SYSTEM Test Reader
  (* Version 1.0, 2005-06-27, Goran Cengic, Chalmers *)
  DEVICE Test Device : DeviceType_not_used
    RESOURCE TestResource : ResourceType_not_used
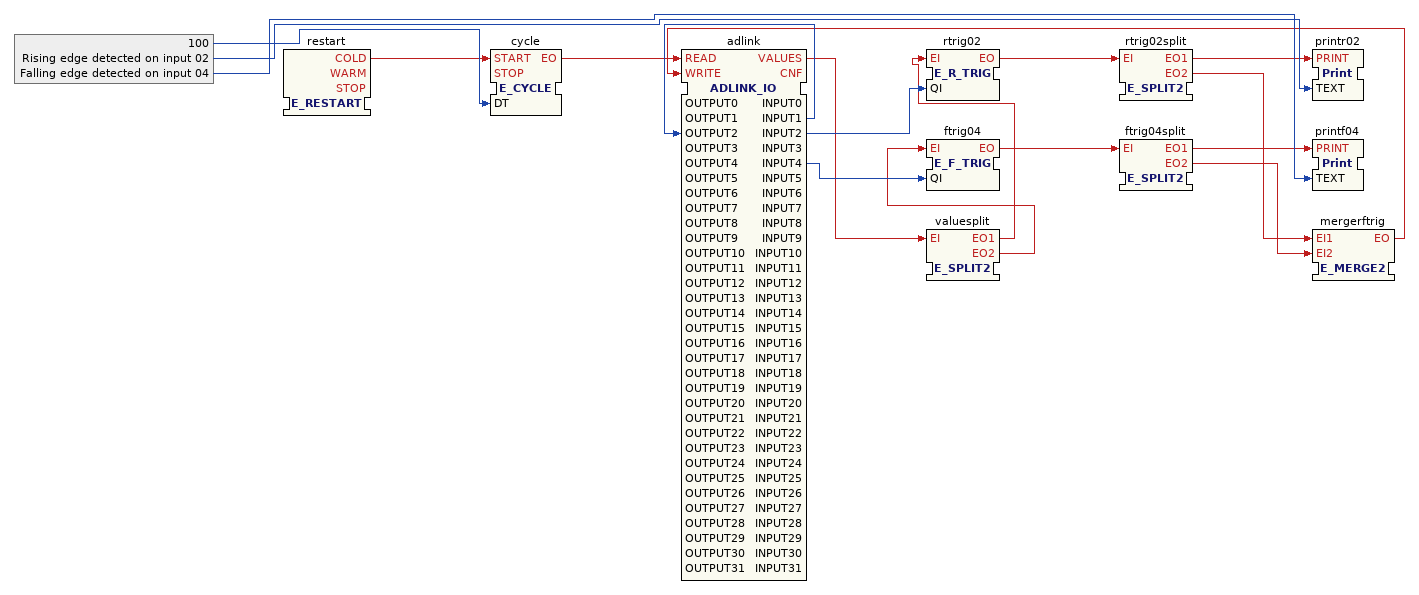
      FBS
        restart : E_RESTART;
        cycle : E_CYCLE;
        adlink : ADLINK_IO;
        rtrig02 : E_R_TRIG;
        ftrig04 : E_F_TRIG;
        valuesplit : E_SPLIT2;
        rtrig02split : E_SPLIT2;
        ftrig04split : E_SPLIT2;
        printr02 : Print;
        printf04 : Print;
        mergerftrig : E_MERGE2;
      END_FBS
      EVENT_CONNECTIONS
        restart.COLD TO cycle.START;
        cycle.EO TO adlink.READ;
        adlink.VALUES TO valuesplit.EI;
        valuesplit.EO1 TO rtrig02.EI;
        valuesplit.EO2 TO ftrig04.EI;
        rtrig02.EO TO rtrig02split.EI;
        ftrig04.EO TO ftrig04split.EI;
        rtrig02split.EO1 TO printr02.PRINT;
        rtrig02split.EO2 TO mergerftrig.EI1;
        ftrig04split.EO1 TO printf04.PRINT;
        ftrig04split.EO2 TO mergerftrig.EI2;
        mergerftrig.EO TO adlink.WRITE;
      END_CONNECTIONS
      DATA_CONNECTIONS
        100 TO cycle.DT;
        adlink.INPUT2 TO rtrig02.QI;
        adlink.INPUT4 TO ftrig04.QI;
        adlink.INPUT1 TO adlink.OUTPUT2;
        Rising edge detected on input 02 TO printr02.TEXT;
        Falling edge detected on input 04 TO printf04.TEXT;
      END_CONNECTIONS
    END_RESOURCE
  END_DEVICE
END_SYSTEM
